{attribute 'GeneratedUsingTerminal: ER6002-0002-0022'}
{attribute addProperty BoxType "ER6002-0002-0022"}
{attribute addProperty Id "CtrlAT %Q*UINT2Data_OutAT %Q*ARRAY[0..21] OF USINT22"}
{attribute addProperty CRC "875731620"}
{attribute addProperty Size "24"}
TYPE COM_RxPDO_Map_Outputs_Channel_5D00B5E7 :
STRUCT
	{attribute addProperty Name "Ctrl"}
	Ctrl AT %Q* : UINT;
	{attribute addProperty Name "Data_Out"}
	Data_Out AT %Q* : ARRAY[0..21] OF USINT;
END_STRUCT
END_TYPE

(* stored: Version 1.2.0.0, ProductVersion 3.1.4024.9
   DUT COM_RxPDO_Map_Outputs_Channel_5D00B5E7: Id {55a7f64f-7e80-45d1-80fb-b476ef9dea68} *)
